PROGRAM pouStation3
VAR
	stationMode: FB_Mode;
	tCalcNumberOfPages: REAL;
	ceil: REAL;
	PartBuild: FB_PartBuild;
	retvall: UDINT;
	// TODO
	tPartPresent: BOOL;
END_VAR

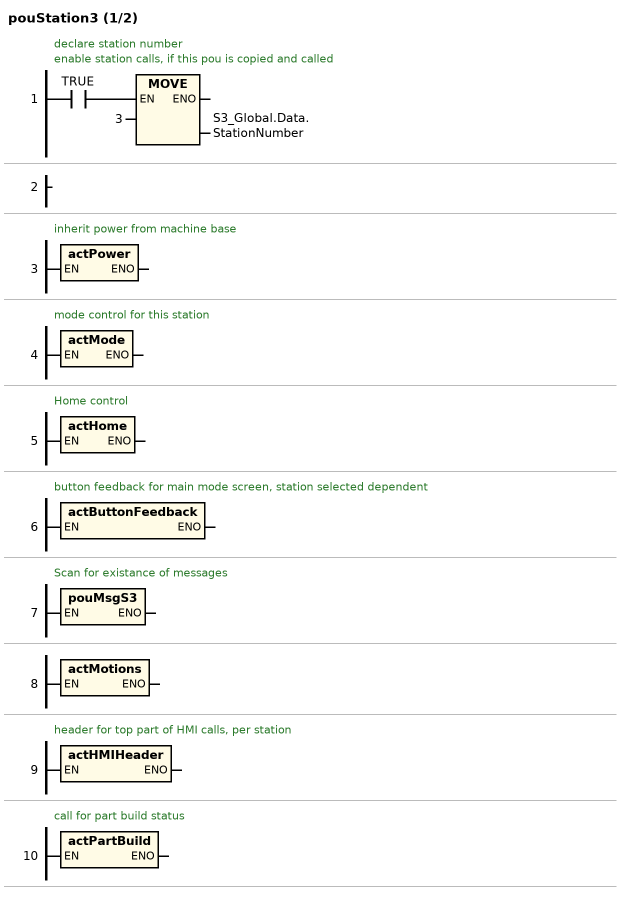
// NETWORK 1
// declare station number
// enable station calls, if this pou is copied and called
S3_Global.Data.StationNumber := 3;

// NETWORK 2

// NETWORK 3
// inherit power from machine base
actPower();

// NETWORK 4
// mode control for this station
actMode();

// NETWORK 5
// Home control
actHome();

// NETWORK 6
// button feedback for main mode screen, station selected dependent
actButtonFeedback();

// NETWORK 7
// Scan for existance of messages
pouMsgS3();

// NETWORK 8
actMotions();

// NETWORK 9
// header for top part of HMI calls, per station
actHMIHeader();

// NETWORK 10
// call for part build status
actPartBuild();

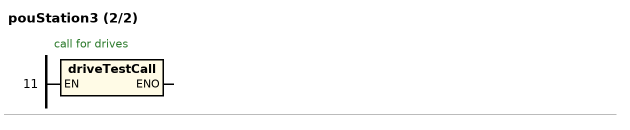
// NETWORK 11
// call for drives
driveTestCall();

ACTION actButtonFeedback:
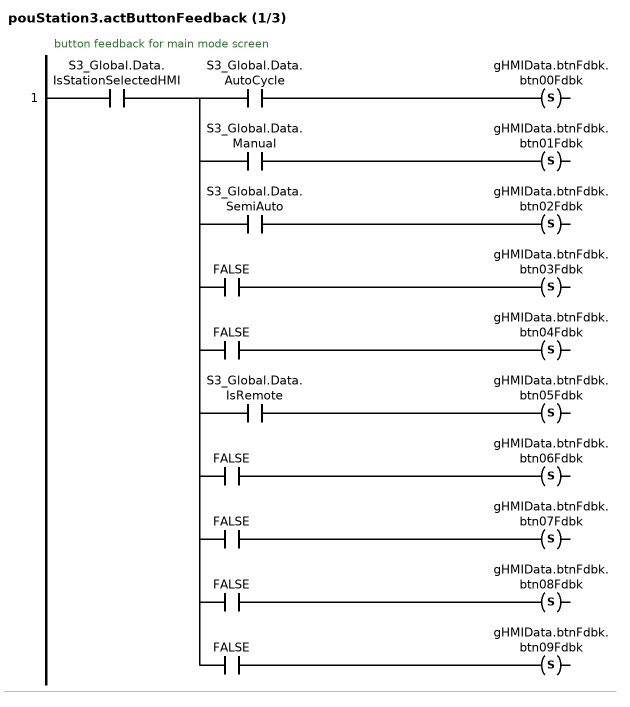
// NETWORK 1
// button feedback for main mode screen
gHMIData.btnFdbk.btn00Fdbk S= S3_Global.Data.IsStationSelectedHMI AND S3_Global.Data.AutoCycle;
gHMIData.btnFdbk.btn01Fdbk S= S3_Global.Data.IsStationSelectedHMI AND S3_Global.Data.Manual;
gHMIData.btnFdbk.btn02Fdbk S= S3_Global.Data.IsStationSelectedHMI AND S3_Global.Data.SemiAuto;
gHMIData.btnFdbk.btn03Fdbk S= S3_Global.Data.IsStationSelectedHMI AND FALSE;
gHMIData.btnFdbk.btn04Fdbk S= S3_Global.Data.IsStationSelectedHMI AND FALSE;
gHMIData.btnFdbk.btn05Fdbk S= S3_Global.Data.IsStationSelectedHMI AND S3_Global.Data.IsRemote;
gHMIData.btnFdbk.btn06Fdbk S= S3_Global.Data.IsStationSelectedHMI AND FALSE;
gHMIData.btnFdbk.btn07Fdbk S= S3_Global.Data.IsStationSelectedHMI AND FALSE;
gHMIData.btnFdbk.btn08Fdbk S= S3_Global.Data.IsStationSelectedHMI AND FALSE;
gHMIData.btnFdbk.btn09Fdbk S= S3_Global.Data.IsStationSelectedHMI AND FALSE;

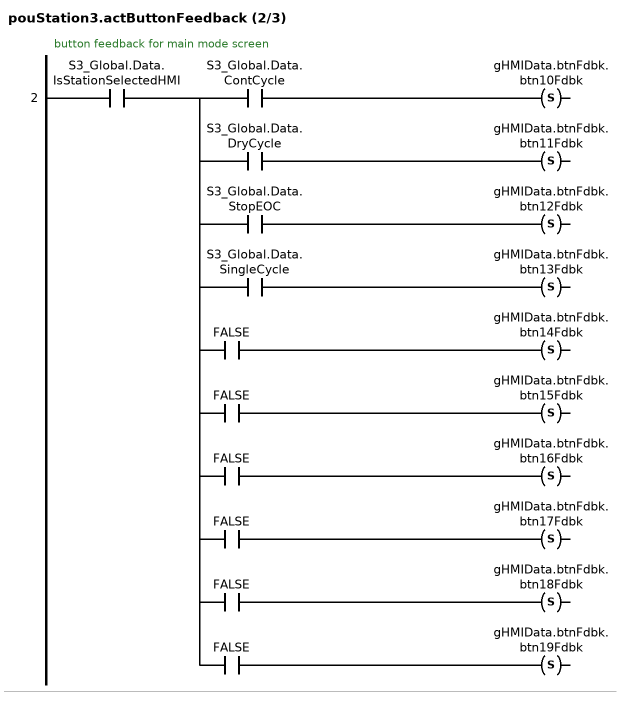
// NETWORK 2
// button feedback for main mode screen
gHMIData.btnFdbk.btn10Fdbk S= S3_Global.Data.IsStationSelectedHMI AND S3_Global.Data.ContCycle;
gHMIData.btnFdbk.btn11Fdbk S= S3_Global.Data.IsStationSelectedHMI AND S3_Global.Data.DryCycle;
gHMIData.btnFdbk.btn12Fdbk S= S3_Global.Data.IsStationSelectedHMI AND S3_Global.Data.StopEOC;
gHMIData.btnFdbk.btn13Fdbk S= S3_Global.Data.IsStationSelectedHMI AND S3_Global.Data.SingleCycle;
gHMIData.btnFdbk.btn14Fdbk S= S3_Global.Data.IsStationSelectedHMI AND FALSE;
gHMIData.btnFdbk.btn15Fdbk S= S3_Global.Data.IsStationSelectedHMI AND FALSE;
gHMIData.btnFdbk.btn16Fdbk S= S3_Global.Data.IsStationSelectedHMI AND FALSE;
gHMIData.btnFdbk.btn17Fdbk S= S3_Global.Data.IsStationSelectedHMI AND FALSE;
gHMIData.btnFdbk.btn18Fdbk S= S3_Global.Data.IsStationSelectedHMI AND FALSE;
gHMIData.btnFdbk.btn19Fdbk S= S3_Global.Data.IsStationSelectedHMI AND FALSE;

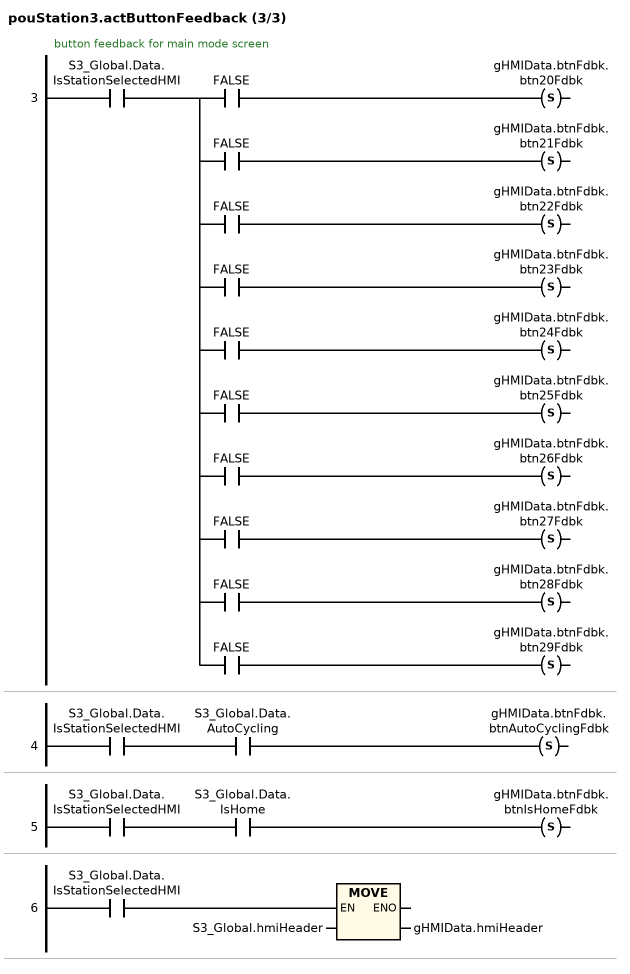
// NETWORK 3
// button feedback for main mode screen
gHMIData.btnFdbk.btn20Fdbk S= S3_Global.Data.IsStationSelectedHMI AND FALSE;
gHMIData.btnFdbk.btn21Fdbk S= S3_Global.Data.IsStationSelectedHMI AND FALSE;
gHMIData.btnFdbk.btn22Fdbk S= S3_Global.Data.IsStationSelectedHMI AND FALSE;
gHMIData.btnFdbk.btn23Fdbk S= S3_Global.Data.IsStationSelectedHMI AND FALSE;
gHMIData.btnFdbk.btn24Fdbk S= S3_Global.Data.IsStationSelectedHMI AND FALSE;
gHMIData.btnFdbk.btn25Fdbk S= S3_Global.Data.IsStationSelectedHMI AND FALSE;
gHMIData.btnFdbk.btn26Fdbk S= S3_Global.Data.IsStationSelectedHMI AND FALSE;
gHMIData.btnFdbk.btn27Fdbk S= S3_Global.Data.IsStationSelectedHMI AND FALSE;
gHMIData.btnFdbk.btn28Fdbk S= S3_Global.Data.IsStationSelectedHMI AND FALSE;
gHMIData.btnFdbk.btn29Fdbk S= S3_Global.Data.IsStationSelectedHMI AND FALSE;

// NETWORK 4
gHMIData.btnFdbk.btnAutoCyclingFdbk S= S3_Global.Data.IsStationSelectedHMI AND S3_Global.Data.AutoCycling;

// NETWORK 5
gHMIData.btnFdbk.btnIsHomeFdbk S= S3_Global.Data.IsStationSelectedHMI AND S3_Global.Data.IsHome;

// NETWORK 6
IF S3_Global.Data.IsStationSelectedHMI THEN gHMIData.hmiHeader := S3_Global.hmiHeader; END_IF
END_ACTION

ACTION actHMIHeader:
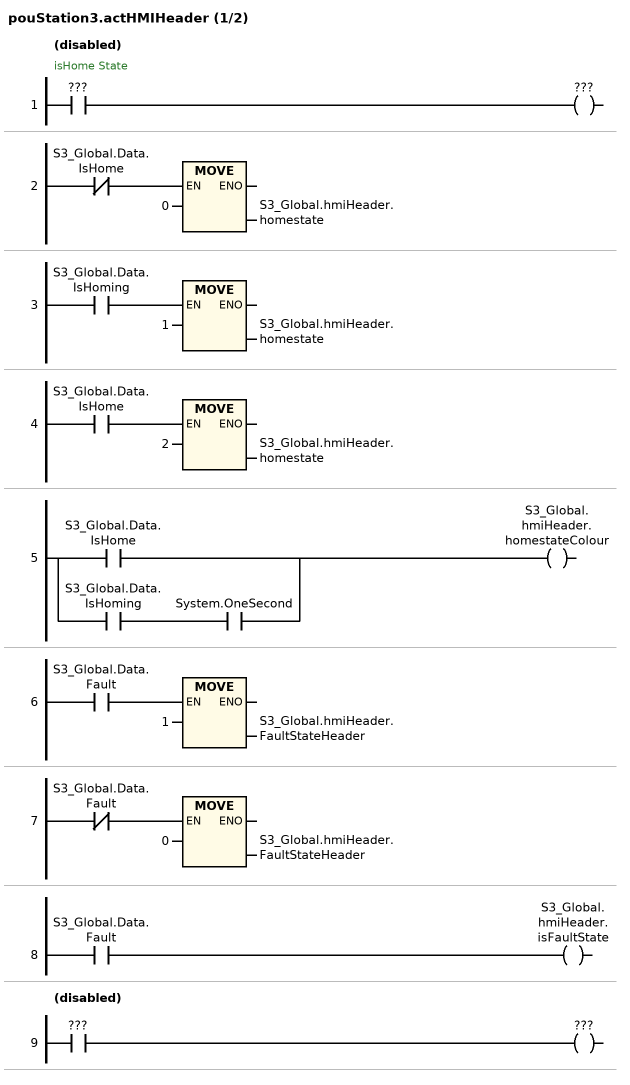
// NETWORK 1 (disabled)
// isHome State
// ??? := ???;

// NETWORK 2
IF NOT S3_Global.Data.IsHome THEN S3_Global.hmiHeader.homestate := 0; END_IF

// NETWORK 3
IF S3_Global.Data.IsHoming THEN S3_Global.hmiHeader.homestate := 1; END_IF

// NETWORK 4
IF S3_Global.Data.IsHome THEN S3_Global.hmiHeader.homestate := 2; END_IF

// NETWORK 5
S3_Global.hmiHeader.homestateColour := S3_Global.Data.IsHome OR S3_Global.Data.IsHoming AND System.OneSecond;

// NETWORK 6
IF S3_Global.Data.Fault THEN S3_Global.hmiHeader.FaultStateHeader := 1; END_IF

// NETWORK 7
IF NOT S3_Global.Data.Fault THEN S3_Global.hmiHeader.FaultStateHeader := 0; END_IF

// NETWORK 8
S3_Global.hmiHeader.isFaultState := S3_Global.Data.Fault;

// NETWORK 9 (disabled)
// ??? := ???;

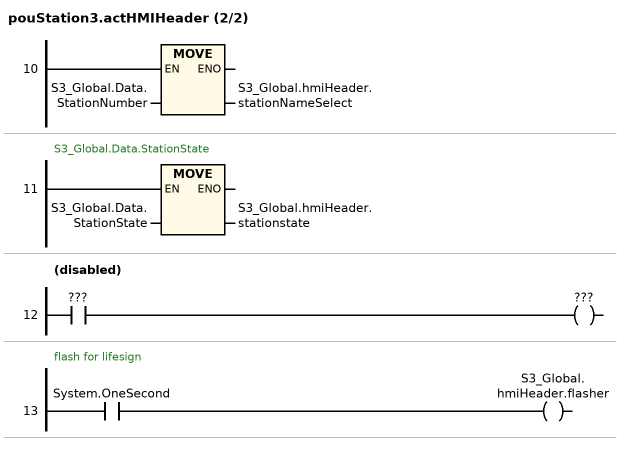
// NETWORK 10
S3_Global.hmiHeader.stationNameSelect := S3_Global.Data.StationNumber;

// NETWORK 11
// S3_Global.Data.StationState
S3_Global.hmiHeader.stationstate := S3_Global.Data.StationState;

// NETWORK 12 (disabled)
// ??? := ???;

// NETWORK 13
// flash for lifesign
S3_Global.hmiHeader.flasher := System.OneSecond;
END_ACTION

ACTION actHome:
//Set home status for station

IF 
//are all motions returned
S3_01_Motion_01_01.Motion.qReturnDepth AND
S3_01_Motion_01_02.Motion.qReturnDepth AND
S3_01_Motion_01_03.Motion.qReturnDepth AND
S3_01_Motion_01_04.Motion.qReturnDepth AND
S3_01_Motion_01_05.Motion.qReturnDepth AND
S3_01_Motion_01_06.Motion.qReturnDepth

	THEN
		//set IsHome value for station
		S3_Global.Data.IsHome := TRUE;
	ELSE
		S3_Global.Data.IsHome := FALSE;
END_IF
END_ACTION

ACTION actMaxNumStationPages:
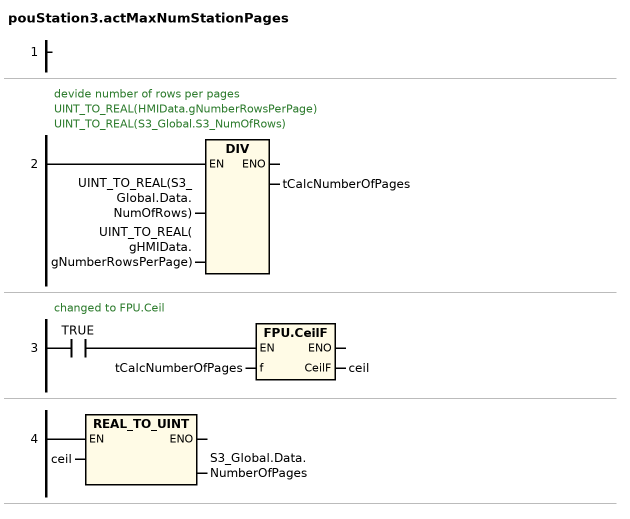
// NETWORK 1

// NETWORK 2
// devide number of rows per pages
// UINT_TO_REAL(HMIData.gNumberRowsPerPage)
// UINT_TO_REAL(S3_Global.S3_NumOfRows)
tCalcNumberOfPages := (UINT_TO_REAL(S3_Global.Data.NumOfRows)) / (UINT_TO_REAL(gHMIData.gNumberRowsPerPage));

// NETWORK 3
// changed to FPU.Ceil
ceil := FPU.CeilF(f := tCalcNumberOfPages);

// NETWORK 4
S3_Global.Data.NumberOfPages := REAL_TO_UINT(ceil);
END_ACTION

ACTION actMode:
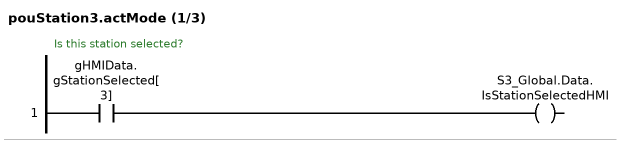
// NETWORK 1
// Is this station selected?
S3_Global.Data.IsStationSelectedHMI := gHMIData.gStationSelected[3];

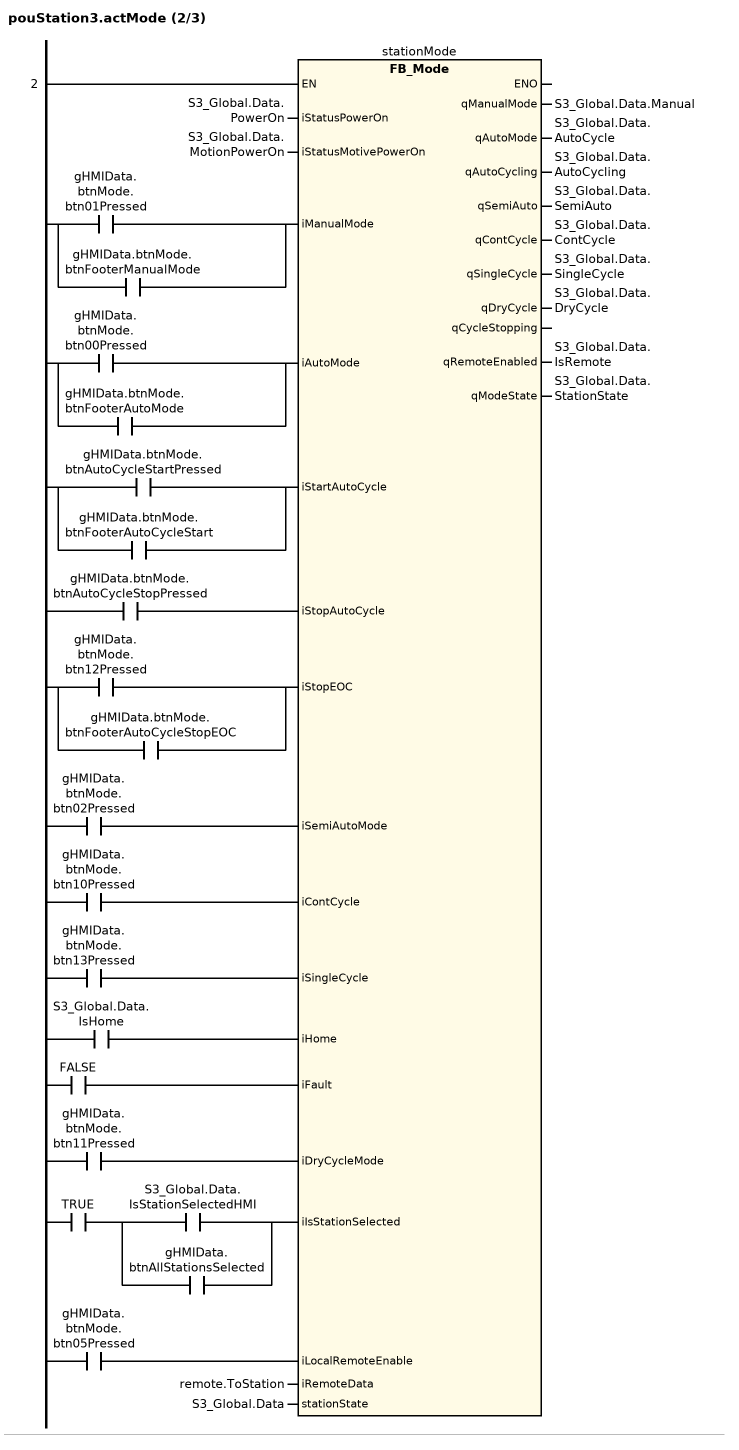
// NETWORK 2
stationMode(
    iStatusPowerOn := S3_Global.Data.PowerOn,
    iStatusMotivePowerOn := S3_Global.Data.MotionPowerOn,
    iManualMode := gHMIData.btnMode.btn01Pressed OR gHMIData.btnMode.btnFooterManualMode,
    iAutoMode := gHMIData.btnMode.btn00Pressed OR gHMIData.btnMode.btnFooterAutoMode,
    iStartAutoCycle := gHMIData.btnMode.btnAutoCycleStartPressed OR gHMIData.btnMode.btnFooterAutoCycleStart,
    iStopAutoCycle := gHMIData.btnMode.btnAutoCycleStopPressed,
    iStopEOC := gHMIData.btnMode.btn12Pressed OR gHMIData.btnMode.btnFooterAutoCycleStopEOC,
    iSemiAutoMode := gHMIData.btnMode.btn02Pressed,
    iContCycle := gHMIData.btnMode.btn10Pressed,
    iSingleCycle := gHMIData.btnMode.btn13Pressed,
    iHome := S3_Global.Data.IsHome,
    iFault := FALSE,
    iDryCycleMode := gHMIData.btnMode.btn11Pressed,
    iIsStationSelected := TRUE AND (S3_Global.Data.IsStationSelectedHMI OR gHMIData.btnAllStationsSelected),
    iLocalRemoteEnable := gHMIData.btnMode.btn05Pressed,
    iRemoteData := remote.ToStation,
    stationState := S3_Global.Data,
    qManualMode => S3_Global.Data.Manual,
    qAutoMode => S3_Global.Data.AutoCycle,
    qAutoCycling => S3_Global.Data.AutoCycling,
    qSemiAuto => S3_Global.Data.SemiAuto,
    qContCycle => S3_Global.Data.ContCycle,
    qSingleCycle => S3_Global.Data.SingleCycle,
    qDryCycle => S3_Global.Data.DryCycle,
    qRemoteEnabled => S3_Global.Data.IsRemote,
    qModeState => S3_Global.Data.StationState); // FB_Mode

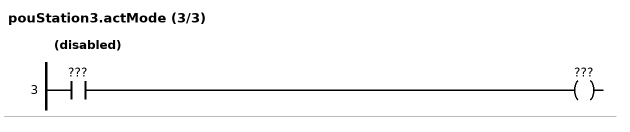
// NETWORK 3 (disabled)
// ??? := ???;
END_ACTION

ACTION actMotions:
//station 1 = 10000 index


//init number of rows
S3_Global.Data.NumOfRows := 0;

//page 1
S3_01_Motion_01_01();
S3_01_Motion_01_02();
S3_01_Motion_01_03();
S3_01_Motion_01_04();
S3_01_Motion_01_05();
S3_01_Motion_01_06();

//page 2
S3_01_Motion_02_07();
S3_01_Motion_02_08();
S3_01_Motion_02_09();
S3_01_Motion_02_10();
S3_01_Motion_02_11();
S3_01_Motion_02_12();

//page 3
S3_01_Motion_03_13();
S3_01_Motion_03_14();
S3_01_Motion_03_15();
S3_01_Motion_03_16();
S3_01_Motion_03_17();
S3_01_Motion_03_18();

//page 4
S3_01_Motion_04_19();
S3_01_Motion_04_20();
S3_01_Motion_04_21();
S3_01_Motion_04_22();
S3_01_Motion_04_23();
S3_01_Motion_04_24();

//page 5
S3_01_Motion_05_25();
S3_01_Motion_05_26();
S3_01_Motion_05_27();
S3_01_Motion_05_28();
S3_01_Motion_05_29();
S3_01_Motion_05_30();

//page 6
S3_01_Motion_06_31();
S3_01_Motion_06_32();
S3_01_Motion_06_33();
S3_01_Motion_06_34();
S3_01_Motion_06_35();
S3_01_Motion_06_36();

//must be called after motionRow calls
actMaxNumStationPages();
END_ACTION

ACTION actPartBuild:
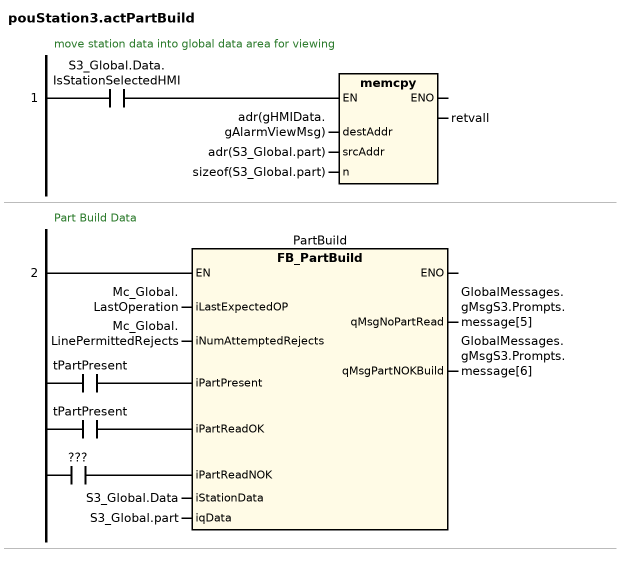
// NETWORK 1
// move station data into global data area for viewing
IF S3_Global.Data.IsStationSelectedHMI THEN
    retvall := memcpy(destAddr := adr(gHMIData.gAlarmViewMsg), srcAddr := adr(S3_Global.part), n := sizeof(S3_Global.part));
END_IF

// NETWORK 2
// Part Build Data
PartBuild(
    iLastExpectedOP := Mc_Global.LastOperation,
    iNumAttemptedRejects := Mc_Global.LinePermittedRejects,
    iPartPresent := tPartPresent,
    iPartReadOK := tPartPresent,
    iStationData := S3_Global.Data,
    iqData := S3_Global.part,
    qMsgNoPartRead => GlobalMessages.gMsgS3.Prompts.message[5],
    qMsgPartNOKBuild => GlobalMessages.gMsgS3.Prompts.message[6]); // FB_PartBuild
END_ACTION

ACTION actPower:
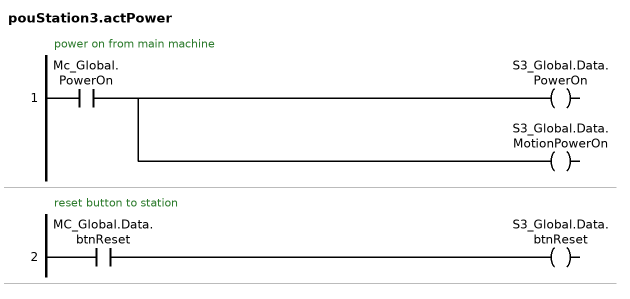
// NETWORK 1
// power on from main machine
S3_Global.Data.PowerOn := Mc_Global.PowerOn;
S3_Global.Data.MotionPowerOn := Mc_Global.PowerOn;

// NETWORK 2
// reset button to station
S3_Global.Data.btnReset := MC_Global.Data.btnReset;
END_ACTION

END_PROGRAM

(* stored: Version 1.1.0.1, ProductVersion 3.1.4024.12
   POU pouStation3: Id {306f601d-e281-4979-9ee6-ccc9093629d3}, SpecialFunc None
   Action actButtonFeedback: Id {dda92a0a-fb1d-41aa-90a2-fa2861dd7530}
   Action actHMIHeader: Id {0ce05a8d-1312-43d8-b8bc-65698172366f}
   Action actHome: Id {c4b50758-b2c2-4fca-935b-f49183e159ed}
   Action actMaxNumStationPages: Id {e7e4958e-9f9a-40ca-8a5d-0419e91ea374}
   Action actMode: Id {5b654011-3f2f-45de-a801-d3e94fb0bba3}
   Action actMotions: Id {e5a7aed3-c679-4a7e-89c9-d64f7eab8660}
   Action actPartBuild: Id {1bfe00d2-d5b0-4c2f-b8c6-7bd73c21f899}
   Action actPower: Id {44d22370-b8e0-4c00-ade3-add7335aab22} *)
